Fanuc KAREL source: kt00042.KL

-- PROVISIONAL review KL for V940-1; original PC SHA256 18cc3394eb18ea04a58c20b7f0ee86bee987b0b83e67fb3c983b81c90145d296
-- Incomplete behavior may be omitted. Consult companion uncertainty JSON. Do not deploy.
PROGRAM KT00042
%NOLOCKGROUP
VAR
  R1 : REAL
  I2 : INTEGER
  OUT : REAL
BEGIN
  -- V9_ZERO_TABLE_METADATA_HINT layout=0001; no indexed target words; source/name/runtime held
  -- UNRESOLVED_PC offsets 5-16; opcodes 2E,23
  -- UNRESOLVED_PC offsets 21-32; opcodes 2E,23
  -- UNRESOLVED_PC offsets 37-57; opcodes 21,21,64,6A,23
  -- UNRESOLVED_PC offsets 62-66; opcodes 7F
END KT00042
